Staubli VAL3: loadmaster3.pgx

program loadmaster3(string x_sMasterFile3 (dimensions=1))
begin
  if master:libLoad(x_sMasterFile3)<0
    popUpMsg("nO ok")
  endIf
  frmaster[3].trsf=master:tTool.trsf
  //取个数
  nsize[3]=size(master:ptRoutingPath)
  //存个数
  resize(pdemo3,1,nsize[3])
  //保存程序
  master:libSave()
end
